INTERFACE I_DemoStep EXTENDS I_Cyclic

METHOD CyclicLogic
END_METHOD

{attribute 'monitoring' := 'call'}
PROPERTY Done : BOOL
GET
END_GET
END_PROPERTY

METHOD Reset : BOOL
VAR_INPUT
END_VAR
END_METHOD

END_INTERFACE

(* stored: Version 1.1.0.1, ProductVersion 3.1.4026.20
   Itf I_DemoStep: Id {9e853b84-91fd-4f0b-930f-fa0ad335ed40}
   Method CyclicLogic: Id {bfa14678-00b4-4747-bae9-f276926d6e15}
   Property Done: Id {d73c1b49-1ed5-45a3-ba89-7b20f42b703d}
   Get Get: Id {63a6f64c-4b92-489f-857c-3d4086495c8f}
   Method Reset: Id {f1c0cf23-6a21-4106-ac5c-20b449a6242c} *)
